// TwinCAT 3 PLC project UnitTests
// Title: Unit Tests for Simple Unit test Lib
// Company: Red Rock Controls Limited
// Author: R Christopher
// ProjectVersion: 1.0.0.0
// ProgramVersion: 3.1.4023.0
// libraries:
//   Tc2_Standard, * (Beckhoff Automation GmbH)
//   Tc2_System, * (Beckhoff Automation GmbH)
//   Tc3_Module, * (Beckhoff Automation GmbH)
//   tcl_SimpleUnitTestLibrary, * (Red Rock Controls Limited)
//   tcl_StringUtils, * (Red Rock Controls Limited)
// project tree:
//   / GlobalTextList.TcGTLO, Visualization Manager.TcVMO (not stored), VISU_TASK.TcTTO
//   GVLs/ UnitTests.TcGVL
//   POUs/ PB_TestRunner.TcPOU
//   POUs/Unit Tests/Assertion Tests/ Test_AssertEquals_BLOB_SizeDiffers.TcPOU, Test_AssertEquals_BLOB_TypeClassDiffers.TcPOU, Test_AssertEquals_BLOB_TypeContentDiffers.TcPOU, Test_AssertEquals_BOOL.TcPOU, Test_AssertEquals_BYTE.TcPOU, Test_AssertEquals_DINT.TcPOU, Test_AssertEquals_DWORD.TcPOU, Test_AssertEquals_INT.TcPOU, Test_AssertEquals_INTERFACE.TcPOU, Test_AssertEquals_LINT.TcPOU, Test_AssertEquals_LREAL.TcPOU, Test_AssertEquals_PVOID.TcPOU, Test_AssertEquals_REAL.TcPOU, Test_AssertEquals_STRING.TcPOU, Test_AssertEquals_UDINT.TcPOU, Test_AssertEquals_UINT.TcPOU, Test_AssertEquals_ULINT.TcPOU, Test_AssertEquals_WORD.TcPOU
//   POUs/Unit Tests/Fixtures/ I_ExampleInterface.TcIO, T_ExampleInterfaceImplementation.TcPOU
//   POUs/Unit Tests/Mocks/ T_AssertionListenerMock.TcPOU
//   POUs/Unit Tests/UnitTestBase Tests/ Test_setTestName_setsTestName.TcPOU, T_UnitTestUnderTest.TcPOU
//   Tasks/ MAIN.TcPOU, PlcTask.TcTTO
//   VISUs/ Visualization.TcVIS
// (motion and I/O tree: see PLC project tcl_simpleunittestlibrary)
// real-time tasks:
//   TASK PlcTask: cycle T#10ms, priority 20, ADS port 351
//   TASK VISU_TASK: cycle T#200000us, priority 30, ADS port 350

CONFIGURATION UnitTests
    RESOURCE PLC ON TwinCAT3
        TASK PlcTask(INTERVAL := T#10ms, PRIORITY := 20);
        TASK VISU_TASK(INTERVAL := T#200000us, PRIORITY := 30);
        PROGRAM MAIN WITH PlcTask : MAIN;
        PROGRAM VisuElems_Visu_Prg WITH VISU_TASK : VisuElems.Visu_Prg;
    END_RESOURCE
END_CONFIGURATION

// ---- GVLs/UnitTests.TcGVL
{attribute 'qualified_only'}
VAR_GLOBAL
    TestFrameworkTests : T_TestSuite;

    Test_AssertEquals_BOOL      : Test_AssertEquals_BOOL        (TestSuite := TestFrameworkTests);
    Test_AssertEquals_BYTE      : Test_AssertEquals_BYTE        (TestSuite := TestFrameworkTests);
    Test_AssertEquals_DINT      : Test_AssertEquals_DINT        (TestSuite := TestFrameworkTests);
    Test_AssertEquals_INT       : Test_AssertEquals_INT         (TestSuite := TestFrameworkTests);
    Test_AssertEquals_INTERFACE : Test_AssertEquals_INTERFACE   (TestSuite := TestFrameworkTests);
    Test_AssertEquals_LINT      : Test_AssertEquals_LINT        (TestSuite := TestFrameworkTests);
    Test_AssertEquals_LREAL     : Test_AssertEquals_LREAL       (TestSuite := TestFrameworkTests);
    Test_AssertEquals_PVOID     : Test_AssertEquals_PVOID       (TestSuite := TestFrameworkTests);
    Test_AssertEquals_REAL      : Test_AssertEquals_REAL        (TestSuite := TestFrameworkTests);
    Test_AssertEquals_STRING    : Test_AssertEquals_STRING      (TestSuite := TestFrameworkTests);
    Test_AssertEquals_UDINT     : Test_AssertEquals_UDINT       (TestSuite := TestFrameworkTests);
    Test_AssertEquals_UINT      : Test_AssertEquals_UINT        (TestSuite := TestFrameworkTests);
    Test_AssertEquals_ULINT     : Test_AssertEquals_ULINT       (TestSuite := TestFrameworkTests);  
    Test_AssertEquals_WORD      : Test_AssertEquals_WORD        (TestSuite := TestFrameworkTests);
    Test_AssertEquals_DWORD     : Test_AssertEquals_DWORD       (TestSuite := TestFrameworkTests);
    
    Test_AssertEquals_BLOB_SizeDiffers          : Test_AssertEquals_BLOB_SizeDiffers        (TestSuite := TestFrameworkTests);  
    Test_AssertEquals_BLOB_TypeClassDiffers     : Test_AssertEquals_BLOB_TypeClassDiffers   (TestSuite := TestFrameworkTests);
    Test_AssertEquals_BLOB_TypeContentDiffers   : Test_AssertEquals_BLOB_TypeContentDiffers (TestSuite := TestFrameworkTests);
    
    Test_setTestName_setsTestName : Test_setTestName_setsTestName (TestSuite := TestFrameworkTests);


END_VAR

// ---- POUs/Unit Tests/Fixtures/I_ExampleInterface.TcIO
INTERFACE I_ExampleInterface EXTENDS __SYSTEM.IQueryInterface

END_INTERFACE

// ---- Tasks/MAIN.TcPOU
PROGRAM MAIN
VAR
END_VAR

PB_TestRunner();

END_PROGRAM

// ---- POUs/PB_TestRunner.TcPOU
PROGRAM PB_TestRunner
VAR
    Init : BOOL := TRUE;
    TestRunner : T_TestRunner;
END_VAR

IF Init THEN
    TestRunner.AddTestSuite(UnitTests.TestFrameworkTests);
    Init := FALSE;
END_IF

TestRunner();

END_PROGRAM

// ---- POUs/Unit Tests/Assertion Tests/Test_AssertEquals_BOOL.TcPOU
FUNCTION_BLOCK Test_AssertEquals_BOOL EXTENDS T_UnitTestBase
VAR
    AssertionUnderTest : T_Assertion(AssertionListenerMock);
    AssertionListenerMock : T_AssertionListenerMock;
    BOOL_Variable : BOOL := FALSE;
END_VAR

// Initialise the classes under test (may be repaeting the tests)...
AssertionListenerMock.fb_Init(
    bInitRetains      := FALSE,
	bInCopyCode       := FALSE);
AssertionUnderTest.fb_Init(
    bInitRetains      := FALSE,
	bInCopyCode       := FALSE,
    AssertionListener := AssertionListenerMock);

// Test the assertion...
AssertionUnderTest.AssertEquals_BOOL(
    Expected := TRUE,
    Actual   := BOOL_Variable,
    VariableName := 'BOOL_Variable');
    
// Check the assertion worked...    
Assertion.AssertEquals_BOOL(
    Expected := TRUE,
    Actual   := AssertionListenerMock.AssertionFailed,
    VariableName := 'AssertionListenerMock.AssertionFailed');

// Check the assertion messages...    
Assertion.AssertEquals_STRING(
    Expected := 'AssertEquals_BOOL failed in AssertionListenerMock: Value "BOOL_Variable"',
    Actual   := AssertionListenerMock.AssertionMessage,
    VariableName := 'AssertionListenerMock.AssertionMessage');

Assertion.AssertEquals_STRING(
    Expected := '  Expected = TRUE',
    Actual   := AssertionListenerMock.ExpectedAsString,
    VariableName := 'AssertionListenerMock.ExpectedAsString');

Assertion.AssertEquals_STRING(
    Expected := '  Actual   = FALSE',
    Actual   := AssertionListenerMock.ActualAsString,
    VariableName := 'AssertionListenerMock.ActualAsString');

TestFinished();

END_FUNCTION_BLOCK

// ---- POUs/Unit Tests/Mocks/T_AssertionListenerMock.TcPOU
{attribute 'reflection'}
FUNCTION_BLOCK T_AssertionListenerMock IMPLEMENTS I_AssertionListener
VAR
    {attribute 'instance-path'} 
    {attribute 'no_init'}
    _FullTestName : T_MaxString; // Automatically initialised with the full name of the instance
    _TestName : T_MaxString; 
    _AssertionFailed  : BOOL;
    _AssertionMessage : T_MaxString;
    _ExpectedAsString : T_MaxString;
    _ActualAsString   : T_MaxString;
END_VAR

PROPERTY ActualAsString : T_MaxString
GET
ActualAsString := _ActualAsString;
END_GET
SET
_ActualAsString := ActualAsString;
END_SET
END_PROPERTY

PROPERTY AssertionFailed : BOOL
GET
AssertionFailed := _AssertionFailed;
END_GET
SET
_AssertionFailed := AssertionFailed;
END_SET
END_PROPERTY

PROPERTY AssertionMessage : T_MaxString
GET
AssertionMessage := _AssertionMessage;
END_GET
SET
_AssertionMessage := AssertionMessage;
END_SET
END_PROPERTY

PROPERTY ExpectedAsString : T_MaxString
GET
ExpectedAsString := _ExpectedAsString;
END_GET
SET
_ExpectedAsString := ExpectedAsString;
END_SET
END_PROPERTY

METHOD OnAssertionFailed
VAR_INPUT
    AssertionMessage : T_MaxString;
    ExpectedAsString : T_MaxString;
    ActualAsString   : T_MaxString;
END_VAR
_AssertionFailed   := TRUE;
_AssertionMessage  := AssertionMessage;
_ExpectedAsString := ExpectedAsString;
_ActualAsString := ActualAsString;
END_METHOD

PROPERTY TestName : Tc2_System.T_MaxString
GET
VAR_INST
    StringSplitter : T_StringSplitter;
END_VAR
IF _TestName = '' THEN
   
    StringSplitter.Init(
        Str := _FullTestName,
        Delim1 := '.',
        Delim2 := '');
    
    WHILE StringSplitter.HasMore() DO
        _TestName := StringSplitter.GetNext(); // to get last sub-section
    END_WHILE
   
END_IF

TestName := _TestName;
END_GET
END_PROPERTY

END_FUNCTION_BLOCK

// ---- POUs/Unit Tests/Assertion Tests/Test_AssertEquals_BYTE.TcPOU
FUNCTION_BLOCK Test_AssertEquals_BYTE EXTENDS T_UnitTestBase
VAR
    AssertionUnderTest : T_Assertion(AssertionListenerMock);
    AssertionListenerMock : T_AssertionListenerMock;
    BYTE_Variable : BYTE := 123;
END_VAR

// Initialise the classes under test (may be repaeting the tests)...
AssertionListenerMock.fb_Init(
    bInitRetains      := FALSE,
	bInCopyCode       := FALSE);
AssertionUnderTest.fb_Init(
    bInitRetains      := FALSE,
	bInCopyCode       := FALSE,
    AssertionListener := AssertionListenerMock);

// Test the assertion...
AssertionUnderTest.AssertEquals_BYTE(
    Expected := 234,
    Actual   := BYTE_Variable,
    VariableName := 'BYTE_Variable');
 
// Check the assertion worked...    
Assertion.AssertEquals_BOOL(
    Expected := TRUE,
    Actual   := AssertionListenerMock.AssertionFailed,
    VariableName := 'AssertionListenerMock.AssertionFailed');

// Check the assertion messages...    
Assertion.AssertEquals_STRING(
    Expected := 'AssertEquals_BYTE failed in AssertionListenerMock: Value "BYTE_Variable"',
    Actual   := AssertionListenerMock.AssertionMessage,
    VariableName := 'AssertionListenerMock.AssertionMessage');

Assertion.AssertEquals_STRING(
    Expected := '  Expected = 234',
    Actual   := AssertionListenerMock.ExpectedAsString,
    VariableName := 'AssertionListenerMock.ExpectedAsString');

Assertion.AssertEquals_STRING(
    Expected := '  Actual   = 123',
    Actual   := AssertionListenerMock.ActualAsString,
    VariableName := 'AssertionListenerMock.ActualAsString');

TestFinished();

END_FUNCTION_BLOCK

// ---- POUs/Unit Tests/Assertion Tests/Test_AssertEquals_DINT.TcPOU
FUNCTION_BLOCK Test_AssertEquals_DINT EXTENDS T_UnitTestBase
VAR
    AssertionUnderTest : T_Assertion(AssertionListenerMock);
    AssertionListenerMock : T_AssertionListenerMock;
    DINT_Variable : DINT := 1111;
END_VAR

// Initialise the classes under test (may be repaeting the tests)...
AssertionListenerMock.fb_Init(
    bInitRetains      := FALSE,
	bInCopyCode       := FALSE);
AssertionUnderTest.fb_Init(
    bInitRetains      := FALSE,
	bInCopyCode       := FALSE,
    AssertionListener := AssertionListenerMock);

// Test the assertion...
AssertionUnderTest.AssertEquals_DINT(
    Expected := 2222,
    Actual   := DINT_Variable,
    VariableName := 'DINT_Variable');
    
// Check the assertion worked...    
Assertion.AssertEquals_BOOL(
    Expected := TRUE,
    Actual   := AssertionListenerMock.AssertionFailed,
    VariableName := 'AssertionListenerMock.AssertionFailed');

// Check the assertion messages...    
Assertion.AssertEquals_STRING(
    Expected := 'AssertEquals_DINT failed in AssertionListenerMock: Value "DINT_Variable"',
    Actual   := AssertionListenerMock.AssertionMessage,
    VariableName := 'AssertionListenerMock.AssertionMessage');

Assertion.AssertEquals_STRING(
    Expected := '  Expected = 2222',
    Actual   := AssertionListenerMock.ExpectedAsString,
    VariableName := 'AssertionListenerMock.ExpectedAsString');

Assertion.AssertEquals_STRING(
    Expected := '  Actual   = 1111',
    Actual   := AssertionListenerMock.ActualAsString,
    VariableName := 'AssertionListenerMock.ActualAsString');

TestFinished();

END_FUNCTION_BLOCK

// ---- POUs/Unit Tests/Assertion Tests/Test_AssertEquals_INT.TcPOU
FUNCTION_BLOCK Test_AssertEquals_INT EXTENDS T_UnitTestBase
VAR
    AssertionUnderTest : T_Assertion(AssertionListenerMock);
    AssertionListenerMock : T_AssertionListenerMock;
    INT_Variable : INT := 1111;
END_VAR

// Initialise the classes under test (may be repaeting the tests)...
AssertionListenerMock.fb_Init(
    bInitRetains      := FALSE,
	bInCopyCode       := FALSE);
AssertionUnderTest.fb_Init(
    bInitRetains      := FALSE,
	bInCopyCode       := FALSE,
    AssertionListener := AssertionListenerMock);

// Test the assertion...
AssertionUnderTest.AssertEquals_INT(
    Expected := 2222,
    Actual   := INT_Variable,
    VariableName := 'INT_Variable');
 
// Check the assertion worked...    
Assertion.AssertEquals_BOOL(
    Expected := TRUE,
    Actual   := AssertionListenerMock.AssertionFailed,
    VariableName := 'AssertionListenerMock.AssertionFailed');

// Check the assertion messages...    
Assertion.AssertEquals_STRING(
    Expected := 'AssertEquals_INT failed in AssertionListenerMock: Value "INT_Variable"',
    Actual   := AssertionListenerMock.AssertionMessage,
    VariableName := 'AssertionListenerMock.AssertionMessage');

Assertion.AssertEquals_STRING(
    Expected := '  Expected = 2222',
    Actual   := AssertionListenerMock.ExpectedAsString,
    VariableName := 'AssertionListenerMock.ExpectedAsString');

Assertion.AssertEquals_STRING(
    Expected := '  Actual   = 1111',
    Actual   := AssertionListenerMock.ActualAsString,
    VariableName := 'AssertionListenerMock.ActualAsString');

TestFinished();

END_FUNCTION_BLOCK

// ---- POUs/Unit Tests/Assertion Tests/Test_AssertEquals_INTERFACE.TcPOU
FUNCTION_BLOCK Test_AssertEquals_INTERFACE EXTENDS T_UnitTestBase
VAR
    AssertionUnderTest : T_Assertion(AssertionListenerMock);
    AssertionListenerMock : T_AssertionListenerMock;
    
    ExampleInterfaceImplementation1   : T_ExampleInterfaceImplementation;
    INTERFACE_Variable1 : I_ExampleInterface := ExampleInterfaceImplementation1;
    
    ExampleInterfaceImplementation2   : T_ExampleInterfaceImplementation;
    INTERFACE_Variable2 : I_ExampleInterface := ExampleInterfaceImplementation2;
END_VAR

// Initialise the classes under test (may be repaeting the tests)...
AssertionListenerMock.fb_Init(
    bInitRetains      := FALSE,
	bInCopyCode       := FALSE);
AssertionUnderTest.fb_Init(
    bInitRetains      := FALSE,
	bInCopyCode       := FALSE,
    AssertionListener := AssertionListenerMock);

// Test the assertion...
AssertionUnderTest.AssertEquals_INTERFACE(
    Expected := INTERFACE_Variable1,
    Actual   := INTERFACE_Variable2,
    VariableName := 'INTERFACE_Variable2'); 
    
// Check the assertion worked...    
Assertion.AssertEquals_BOOL(
    Expected := TRUE,
    Actual   := AssertionListenerMock.AssertionFailed,
    VariableName := 'AssertionListenerMock.AssertionFailed');

// Check the assertion messages...    
Assertion.AssertEquals_STRING(
    Expected := 'AssertEquals_INTERFACE failed in AssertionListenerMock: Value "INTERFACE_Variable2"',
    Actual   := AssertionListenerMock.AssertionMessage,
    VariableName := 'AssertionListenerMock.AssertionMessage');

Assertion.AssertEquals_STRING(
    Expected := '  Interfaces Differ',
    Actual   := AssertionListenerMock.ExpectedAsString,
    VariableName := 'AssertionListenerMock.ExpectedAsString');

Assertion.AssertEquals_STRING(
    Expected := '',
    Actual   := AssertionListenerMock.ActualAsString,
    VariableName := 'AssertionListenerMock.ActualAsString');

TestFinished();

END_FUNCTION_BLOCK

// ---- POUs/Unit Tests/Fixtures/T_ExampleInterfaceImplementation.TcPOU
FUNCTION_BLOCK T_ExampleInterfaceImplementation IMPLEMENTS I_ExampleInterface
VAR_INPUT
END_VAR
VAR_OUTPUT
END_VAR
VAR
END_VAR

END_FUNCTION_BLOCK

// ---- POUs/Unit Tests/Assertion Tests/Test_AssertEquals_LINT.TcPOU
FUNCTION_BLOCK Test_AssertEquals_LINT EXTENDS T_UnitTestBase
VAR
    AssertionUnderTest : T_Assertion(AssertionListenerMock);
    AssertionListenerMock : T_AssertionListenerMock;
    LINT_Variable : LINT := 1111;
END_VAR

// Initialise the classes under test (may be repaeting the tests)...
AssertionListenerMock.fb_Init(
    bInitRetains      := FALSE,
	bInCopyCode       := FALSE);
AssertionUnderTest.fb_Init(
    bInitRetains      := FALSE,
	bInCopyCode       := FALSE,
    AssertionListener := AssertionListenerMock);

// Test the assertion...
AssertionUnderTest.AssertEquals_LINT(
    Expected := 2222,
    Actual   := LINT_Variable,
    VariableName := 'LINT_Variable');
 
    
// Check the assertion worked...    
Assertion.AssertEquals_BOOL(
    Expected := TRUE,
    Actual   := AssertionListenerMock.AssertionFailed,
    VariableName := 'AssertionListenerMock.AssertionFailed');

// Check the assertion messages...    
Assertion.AssertEquals_STRING(
    Expected := 'AssertEquals_LINT failed in AssertionListenerMock: Value "LINT_Variable"',
    Actual   := AssertionListenerMock.AssertionMessage,
    VariableName := 'AssertionListenerMock.AssertionMessage');

Assertion.AssertEquals_STRING(
    Expected := '  Expected = 2222',
    Actual   := AssertionListenerMock.ExpectedAsString,
    VariableName := 'AssertionListenerMock.ExpectedAsString');

Assertion.AssertEquals_STRING(
    Expected := '  Actual   = 1111',
    Actual   := AssertionListenerMock.ActualAsString,
    VariableName := 'AssertionListenerMock.ActualAsString');

TestFinished();

END_FUNCTION_BLOCK

// ---- POUs/Unit Tests/Assertion Tests/Test_AssertEquals_LREAL.TcPOU
FUNCTION_BLOCK Test_AssertEquals_LREAL EXTENDS T_UnitTestBase
VAR
    AssertionUnderTest : T_Assertion(AssertionListenerMock);
    AssertionListenerMock : T_AssertionListenerMock;
    LREAL_Variable : LREAL := 1.111;
END_VAR

// Initialise the classes under test (may be repaeting the tests)...
AssertionListenerMock.fb_Init(
    bInitRetains      := FALSE,
	bInCopyCode       := FALSE);
AssertionUnderTest.fb_Init(
    bInitRetains      := FALSE,
	bInCopyCode       := FALSE,
    AssertionListener := AssertionListenerMock);

// Test the assertion...
AssertionUnderTest.AssertEquals_LREAL(
    Expected := 2.222,
    Actual   := LREAL_Variable,
    Delta    := 0.001,
    VariableName := 'LREAL_Variable');
   
// Check the assertion worked...    
Assertion.AssertEquals_BOOL(
    Expected := TRUE,
    Actual   := AssertionListenerMock.AssertionFailed,
    VariableName := 'AssertionListenerMock.AssertionFailed');

// Check the assertion messages...    
Assertion.AssertEquals_STRING(
    Expected := 'AssertEquals_LREAL failed in AssertionListenerMock: Value "LREAL_Variable"',
    Actual   := AssertionListenerMock.AssertionMessage,
    VariableName := 'AssertionListenerMock.AssertionMessage');

Assertion.AssertEquals_STRING(
    Expected := '  Expected = 2.222000',
    Actual   := AssertionListenerMock.ExpectedAsString,
    VariableName := 'AssertionListenerMock.ExpectedAsString');

Assertion.AssertEquals_STRING(
    Expected := '  Actual   = 1.111000',
    Actual   := AssertionListenerMock.ActualAsString,
    VariableName := 'AssertionListenerMock.ActualAsString');

TestFinished();

END_FUNCTION_BLOCK

// ---- POUs/Unit Tests/Assertion Tests/Test_AssertEquals_PVOID.TcPOU
FUNCTION_BLOCK Test_AssertEquals_PVOID EXTENDS T_UnitTestBase
VAR
    AssertionUnderTest : T_Assertion(AssertionListenerMock);
    AssertionListenerMock : T_AssertionListenerMock;
    PVOID_Variable : PVOID := 1111;
END_VAR

// Initialise the classes under test (may be repaeting the tests)...
AssertionListenerMock.fb_Init(
    bInitRetains      := FALSE,
	bInCopyCode       := FALSE);
AssertionUnderTest.fb_Init(
    bInitRetains      := FALSE,
	bInCopyCode       := FALSE,
    AssertionListener := AssertionListenerMock);

// Test the assertion...
AssertionUnderTest.AssertEquals_PVOID(
    Expected := 2222,
    Actual   := PVOID_Variable,
    VariableName := 'PVOID_Variable'); 
    
// Check the assertion worked...    
Assertion.AssertEquals_BOOL(
    Expected := TRUE,
    Actual   := AssertionListenerMock.AssertionFailed,
    VariableName := 'AssertionListenerMock.AssertionFailed');

// Check the assertion messages...    
Assertion.AssertEquals_STRING(
    Expected := 'AssertEquals_PVOID failed in AssertionListenerMock: Value "PVOID_Variable"',
    Actual   := AssertionListenerMock.AssertionMessage,
    VariableName := 'AssertionListenerMock.AssertionMessage');

Assertion.AssertEquals_STRING(
    Expected := '  Expected = 2222',
    Actual   := AssertionListenerMock.ExpectedAsString,
    VariableName := 'AssertionListenerMock.ExpectedAsString');

Assertion.AssertEquals_STRING(
    Expected := '  Actual   = 1111',
    Actual   := AssertionListenerMock.ActualAsString,
    VariableName := 'AssertionListenerMock.ActualAsString');

TestFinished();

END_FUNCTION_BLOCK

// ---- POUs/Unit Tests/Assertion Tests/Test_AssertEquals_REAL.TcPOU
FUNCTION_BLOCK Test_AssertEquals_REAL EXTENDS T_UnitTestBase
VAR
    AssertionUnderTest : T_Assertion(AssertionListenerMock);
    AssertionListenerMock : T_AssertionListenerMock;
    REAL_Variable : REAL := 1.111;
END_VAR

// Initialise the classes under test (may be repaeting the tests)...
AssertionListenerMock.fb_Init(
    bInitRetains      := FALSE,
	bInCopyCode       := FALSE);
AssertionUnderTest.fb_Init(
    bInitRetains      := FALSE,
	bInCopyCode       := FALSE,
    AssertionListener := AssertionListenerMock);

// Test the assertion...
AssertionUnderTest.AssertEquals_REAL(
    Expected := 2.222,
    Actual   := REAL_Variable,
    Delta    := 0.001,
    VariableName := 'REAL_Variable');
  
// Check the assertion worked...    
Assertion.AssertEquals_BOOL(
    Expected := TRUE,
    Actual   := AssertionListenerMock.AssertionFailed,
    VariableName := 'AssertionListenerMock.AssertionFailed');

// Check the assertion messages...    
Assertion.AssertEquals_STRING(
    Expected := 'AssertEquals_REAL failed in AssertionListenerMock: Value "REAL_Variable"',
    Actual   := AssertionListenerMock.AssertionMessage,
    VariableName := 'AssertionListenerMock.AssertionMessage');

Assertion.AssertEquals_STRING(
    Expected := '  Expected = 2.222000',
    Actual   := AssertionListenerMock.ExpectedAsString,
    VariableName := 'AssertionListenerMock.ExpectedAsString');

Assertion.AssertEquals_STRING(
    Expected := '  Actual   = 1.111000',
    Actual   := AssertionListenerMock.ActualAsString,
    VariableName := 'AssertionListenerMock.ActualAsString');

TestFinished();

END_FUNCTION_BLOCK

// ---- POUs/Unit Tests/Assertion Tests/Test_AssertEquals_STRING.TcPOU
FUNCTION_BLOCK Test_AssertEquals_STRING EXTENDS T_UnitTestBase
VAR
    AssertionUnderTest : T_Assertion(AssertionListenerMock);
    AssertionListenerMock : T_AssertionListenerMock;
    STRING_Variable : STRING := 'Cucumber';
END_VAR

// Initialise the classes under test (may be repaeting the tests)...
AssertionListenerMock.fb_Init(
    bInitRetains      := FALSE,
	bInCopyCode       := FALSE);
AssertionUnderTest.fb_Init(
    bInitRetains      := FALSE,
	bInCopyCode       := FALSE,
    AssertionListener := AssertionListenerMock);

// Test the assertion...
AssertionUnderTest.AssertEquals_STRING(
    Expected := 'Radish',
    Actual   := STRING_Variable,
    VariableName := 'STRING_Variable'); 
    
// Check the assertion worked...    
Assertion.AssertEquals_BOOL(
    Expected := TRUE,
    Actual   := AssertionListenerMock.AssertionFailed,
    VariableName := 'AssertionListenerMock.AssertionFailed');

// Check the assertion messages...    
Assertion.AssertEquals_STRING(
    Expected := 'AssertEquals_STRING failed in AssertionListenerMock: Value "STRING_Variable"',
    Actual   := AssertionListenerMock.AssertionMessage,
    VariableName := 'AssertionListenerMock.AssertionMessage');

Assertion.AssertEquals_STRING(
    Expected := '  Expected = Radish',
    Actual   := AssertionListenerMock.ExpectedAsString,
    VariableName := 'AssertionListenerMock.ExpectedAsString');

Assertion.AssertEquals_STRING(
    Expected := '  Actual   = Cucumber',
    Actual   := AssertionListenerMock.ActualAsString,
    VariableName := 'AssertionListenerMock.ActualAsString');

TestFinished();

END_FUNCTION_BLOCK

// ---- POUs/Unit Tests/Assertion Tests/Test_AssertEquals_UDINT.TcPOU
FUNCTION_BLOCK Test_AssertEquals_UDINT EXTENDS T_UnitTestBase
VAR
    AssertionUnderTest : T_Assertion(AssertionListenerMock);
    AssertionListenerMock : T_AssertionListenerMock;
    UDINT_Variable : UDINT := 1111;
END_VAR

// Initialise the classes under test (may be repaeting the tests)...
AssertionListenerMock.fb_Init(
    bInitRetains      := FALSE,
	bInCopyCode       := FALSE);
AssertionUnderTest.fb_Init(
    bInitRetains      := FALSE,
	bInCopyCode       := FALSE,
    AssertionListener := AssertionListenerMock);

// Test the assertion...
AssertionUnderTest.AssertEquals_UDINT(
    Expected := 2222,
    Actual   := UDINT_Variable,
    VariableName := 'UDINT_Variable');
    
// Check the assertion worked...    
Assertion.AssertEquals_BOOL(
    Expected := TRUE,
    Actual   := AssertionListenerMock.AssertionFailed,
    VariableName := 'AssertionListenerMock.AssertionFailed');

// Check the assertion messages...    
Assertion.AssertEquals_STRING(
    Expected := 'AssertEquals_UDINT failed in AssertionListenerMock: Value "UDINT_Variable"',
    Actual   := AssertionListenerMock.AssertionMessage,
    VariableName := 'AssertionListenerMock.AssertionMessage');

Assertion.AssertEquals_STRING(
    Expected := '  Expected = 2222',
    Actual   := AssertionListenerMock.ExpectedAsString,
    VariableName := 'AssertionListenerMock.ExpectedAsString');

Assertion.AssertEquals_STRING(
    Expected := '  Actual   = 1111',
    Actual   := AssertionListenerMock.ActualAsString,
    VariableName := 'AssertionListenerMock.ActualAsString');

TestFinished();

END_FUNCTION_BLOCK

// ---- POUs/Unit Tests/Assertion Tests/Test_AssertEquals_UINT.TcPOU
FUNCTION_BLOCK Test_AssertEquals_UINT EXTENDS T_UnitTestBase
VAR
    AssertionUnderTest : T_Assertion(AssertionListenerMock);
    AssertionListenerMock : T_AssertionListenerMock;
    UINT_Variable : UINT := 1111;
END_VAR

// Initialise the classes under test (may be repaeting the tests)...
AssertionListenerMock.fb_Init(
    bInitRetains      := FALSE,
	bInCopyCode       := FALSE);
AssertionUnderTest.fb_Init(
    bInitRetains      := FALSE,
	bInCopyCode       := FALSE,
    AssertionListener := AssertionListenerMock);

// Test the assertion...
AssertionUnderTest.AssertEquals_UINT(
    Expected := 2222,
    Actual   := UINT_Variable,
    VariableName := 'UINT_Variable');
   
// Check the assertion worked...    
Assertion.AssertEquals_BOOL(
    Expected := TRUE,
    Actual   := AssertionListenerMock.AssertionFailed,
    VariableName := 'AssertionListenerMock.AssertionFailed');

// Check the assertion messages...    
Assertion.AssertEquals_STRING(
    Expected := 'AssertEquals_UINT failed in AssertionListenerMock: Value "UINT_Variable"',
    Actual   := AssertionListenerMock.AssertionMessage,

    VariableName := 'AssertionListenerMock.AssertionMessage');

Assertion.AssertEquals_STRING(
    Expected := '  Expected = 2222',
    Actual   := AssertionListenerMock.ExpectedAsString,
    VariableName := 'AssertionListenerMock.ExpectedAsString');

Assertion.AssertEquals_STRING(
    Expected := '  Actual   = 1111',
    Actual   := AssertionListenerMock.ActualAsString,
    VariableName := 'AssertionListenerMock.ActualAsString');

TestFinished();

END_FUNCTION_BLOCK

// ---- POUs/Unit Tests/Assertion Tests/Test_AssertEquals_ULINT.TcPOU
FUNCTION_BLOCK Test_AssertEquals_ULINT EXTENDS T_UnitTestBase
VAR
    AssertionUnderTest : T_Assertion(AssertionListenerMock);
    AssertionListenerMock : T_AssertionListenerMock;
    ULINT_Variable : ULINT := 1111;
END_VAR

// Initialise the classes under test (may be repaeting the tests)...
AssertionListenerMock.fb_Init(
    bInitRetains      := FALSE,
	bInCopyCode       := FALSE);
AssertionUnderTest.fb_Init(
    bInitRetains      := FALSE,
	bInCopyCode       := FALSE,
    AssertionListener := AssertionListenerMock);

// Test the assertion...
AssertionUnderTest.AssertEquals_ULINT(
    Expected := 2222,
    Actual   := ULINT_Variable,
    VariableName := 'ULINT_Variable');
   
// Check the assertion worked...    
Assertion.AssertEquals_BOOL(
    Expected := TRUE,
    Actual   := AssertionListenerMock.AssertionFailed,
    VariableName := 'AssertionListenerMock.AssertionFailed');

// Check the assertion messages...    
Assertion.AssertEquals_STRING(
    Expected := 'AssertEquals_ULINT failed in AssertionListenerMock: Value "ULINT_Variable"',
    Actual   := AssertionListenerMock.AssertionMessage,
    VariableName := 'AssertionListenerMock.AssertionMessage');

Assertion.AssertEquals_STRING(
    Expected := '  Expected = 2222',
    Actual   := AssertionListenerMock.ExpectedAsString,
    VariableName := 'AssertionListenerMock.ExpectedAsString');

Assertion.AssertEquals_STRING(
    Expected := '  Actual   = 1111',
    Actual   := AssertionListenerMock.ActualAsString,
    VariableName := 'AssertionListenerMock.ActualAsString');

TestFinished();

END_FUNCTION_BLOCK

// ---- POUs/Unit Tests/Assertion Tests/Test_AssertEquals_WORD.TcPOU
FUNCTION_BLOCK Test_AssertEquals_WORD EXTENDS T_UnitTestBase
VAR
    AssertionUnderTest : T_Assertion(AssertionListenerMock);
    AssertionListenerMock : T_AssertionListenerMock;
    WORD_Variable : WORD;
END_VAR

// Initialise the classes under test (may be repaeting the tests)...
AssertionListenerMock.fb_Init(
    bInitRetains      := FALSE,
	bInCopyCode       := FALSE);
AssertionUnderTest.fb_Init(
    bInitRetains      := FALSE,
	bInCopyCode       := FALSE,
    AssertionListener := AssertionListenerMock);

// Test the assertion...
WORD_Variable := 1111;

AssertionUnderTest.AssertEquals_WORD(
    Expected := 2222, // deliberately different to test the assertion
    Actual   := WORD_Variable,
    VariableName := 'WORD_Variable');
 
// Check the assertion worked...    
Assertion.AssertEquals_BOOL(
    Expected := TRUE,
    Actual   := AssertionListenerMock.AssertionFailed,
    VariableName := 'AssertionListenerMock.AssertionFailed');

// Check the assertion messages...    
Assertion.AssertEquals_STRING(
    Expected := 'AssertEquals_WORD failed in AssertionListenerMock: Value "WORD_Variable"',
    Actual   := AssertionListenerMock.AssertionMessage,
    VariableName := 'AssertionListenerMock.AssertionMessage');

Assertion.AssertEquals_STRING(
    Expected := '  Expected = 2222',
    Actual   := AssertionListenerMock.ExpectedAsString,
    VariableName := 'AssertionListenerMock.ExpectedAsString');

Assertion.AssertEquals_STRING(
    Expected := '  Actual   = 1111',
    Actual   := AssertionListenerMock.ActualAsString,
    VariableName := 'AssertionListenerMock.ActualAsString');


TestFinished();

END_FUNCTION_BLOCK

// ---- POUs/Unit Tests/Assertion Tests/Test_AssertEquals_DWORD.TcPOU
FUNCTION_BLOCK Test_AssertEquals_DWORD EXTENDS T_UnitTestBase
VAR
    AssertionUnderTest : T_Assertion(AssertionListenerMock);
    AssertionListenerMock : T_AssertionListenerMock;
    DWORD_Variable : DWORD;
END_VAR

// Initialise the classes under test (may be repaeting the tests)...
AssertionListenerMock.fb_Init(
    bInitRetains      := FALSE,
	bInCopyCode       := FALSE);
AssertionUnderTest.fb_Init(
    bInitRetains      := FALSE,
	bInCopyCode       := FALSE,
    AssertionListener := AssertionListenerMock);

// Test the assertion...
DWORD_Variable := 1111;

AssertionUnderTest.AssertEquals_DWORD(
    Expected := 2222, // deliberately different to test the assertion
    Actual   := DWORD_Variable,
    VariableName := 'DWORD_Variable');
 
    
// Check the assertion worked...    
Assertion.AssertEquals_BOOL(
    Expected := TRUE,
    Actual   := AssertionListenerMock.AssertionFailed,
    VariableName := 'AssertionListenerMock.AssertionFailed');

// Check the assertion messages...    
Assertion.AssertEquals_STRING(
    Expected := 'AssertEquals_DWORD failed in AssertionListenerMock: Value "DWORD_Variable"',
    Actual   := AssertionListenerMock.AssertionMessage,
    VariableName := 'AssertionListenerMock.AssertionMessage');

Assertion.AssertEquals_STRING(
    Expected := '  Expected = 2222',
    Actual   := AssertionListenerMock.ExpectedAsString,
    VariableName := 'AssertionListenerMock.ExpectedAsString');

Assertion.AssertEquals_STRING(
    Expected := '  Actual   = 1111',
    Actual   := AssertionListenerMock.ActualAsString,
    VariableName := 'AssertionListenerMock.ActualAsString');

TestFinished();

END_FUNCTION_BLOCK

// ---- POUs/Unit Tests/Assertion Tests/Test_AssertEquals_BLOB_SizeDiffers.TcPOU
FUNCTION_BLOCK Test_AssertEquals_BLOB_SizeDiffers EXTENDS T_UnitTestBase
VAR
    AssertionUnderTest : T_Assertion(AssertionListenerMock);
    AssertionListenerMock : T_AssertionListenerMock;
    BYTE_Variable : BYTE := 123;
    WORD_Variable : WORD := 456;
END_VAR

// Initialise the classes under test (may be repaeting the tests)...
AssertionListenerMock.fb_Init(
    bInitRetains      := FALSE,
	bInCopyCode       := FALSE);
AssertionUnderTest.fb_Init(
    bInitRetains      := FALSE,
	bInCopyCode       := FALSE,
    AssertionListener := AssertionListenerMock);

// Test the assertion...
AssertionUnderTest.AssertEquals_BLOB(
    Expected := BYTE_Variable,
    Actual   := WORD_Variable,
    VariableName := 'WORD_VariableAsBlob');
 
    
// Check the assertion worked...    
Assertion.AssertEquals_BOOL(
    Expected := TRUE,
    Actual   := AssertionListenerMock.AssertionFailed,
    VariableName := 'AssertionListenerMock.AssertionFailed');

// Check the assertion messages...    
Assertion.AssertEquals_STRING(
    Expected := 'AssertEquals_BLOB failed in AssertionListenerMock: Value "Blob.Size"',
    Actual   := AssertionListenerMock.AssertionMessage,
    VariableName := 'AssertionListenerMock.AssertionMessage');

Assertion.AssertEquals_STRING(
    Expected := '  Expected = 1',
    Actual   := AssertionListenerMock.ExpectedAsString,
    VariableName := 'AssertionListenerMock.ExpectedAsString');

Assertion.AssertEquals_STRING(
    Expected := '  Actual   = 2',
    Actual   := AssertionListenerMock.ActualAsString,
    VariableName := 'AssertionListenerMock.ActualAsString');

TestFinished();

END_FUNCTION_BLOCK

// ---- POUs/Unit Tests/Assertion Tests/Test_AssertEquals_BLOB_TypeClassDiffers.TcPOU
FUNCTION_BLOCK Test_AssertEquals_BLOB_TypeClassDiffers EXTENDS T_UnitTestBase
VAR
    AssertionUnderTest : T_Assertion(AssertionListenerMock);
    AssertionListenerMock : T_AssertionListenerMock;
    
    // Sizes are the same, but TypeClass differs...
    INT_Variable  : INT  := 123;
    WORD_Variable : WORD := 123;
END_VAR

// Initialise the classes under test (may be repaeting the tests)...
AssertionListenerMock.fb_Init(
    bInitRetains      := FALSE,
	bInCopyCode       := FALSE);
AssertionUnderTest.fb_Init(
    bInitRetains      := FALSE,
	bInCopyCode       := FALSE,
    AssertionListener := AssertionListenerMock);

// Test the assertion...
AssertionUnderTest.AssertEquals_BLOB(
    Expected := INT_Variable,
    Actual   := WORD_Variable,
    VariableName := 'WORD_VariableAsBlob');
 
// Check the assertion worked...    
Assertion.AssertEquals_BOOL(
    Expected := TRUE,
    Actual   := AssertionListenerMock.AssertionFailed,
    VariableName := 'AssertionListenerMock.AssertionFailed');

// Check the assertion messages...    
Assertion.AssertEquals_STRING(
    Expected := 'AssertEquals_BLOB failed in AssertionListenerMock: Value "Blob.TypeClass"',
    Actual   := AssertionListenerMock.AssertionMessage,
    VariableName := 'AssertionListenerMock.AssertionMessage');

Assertion.AssertEquals_STRING(
    Expected := '  Expected = INT',
    Actual   := AssertionListenerMock.ExpectedAsString,
    VariableName := 'AssertionListenerMock.ExpectedAsString');

Assertion.AssertEquals_STRING(
    Expected := '  Actual   = WORD',
    Actual   := AssertionListenerMock.ActualAsString,
    VariableName := 'AssertionListenerMock.ActualAsString');

TestFinished();

END_FUNCTION_BLOCK

// ---- POUs/Unit Tests/Assertion Tests/Test_AssertEquals_BLOB_TypeContentDiffers.TcPOU
FUNCTION_BLOCK Test_AssertEquals_BLOB_TypeContentDiffers EXTENDS T_UnitTestBase
VAR
    AssertionUnderTest : T_Assertion(AssertionListenerMock);
    AssertionListenerMock : T_AssertionListenerMock;
    
    // Sizes are the same, but TypeClass differs...
    INT_Variable  : WORD := 123;
    WORD_Variable : WORD := 124;
END_VAR

// Initialise the classes under test (may be repaeting the tests)...
AssertionListenerMock.fb_Init(
    bInitRetains      := FALSE,
	bInCopyCode       := FALSE);
AssertionUnderTest.fb_Init(
    bInitRetains      := FALSE,
	bInCopyCode       := FALSE,
    AssertionListener := AssertionListenerMock);

// Test the assertion...
AssertionUnderTest.AssertEquals_BLOB(
    Expected := INT_Variable,
    Actual   := WORD_Variable,
    VariableName := 'WORD_VariableAsBlob');
 
// Check the assertion worked...    
Assertion.AssertEquals_BOOL(
    Expected := TRUE,
    Actual   := AssertionListenerMock.AssertionFailed,
    VariableName := 'AssertionListenerMock.AssertionFailed');

// Check the assertion messages...    
Assertion.AssertEquals_STRING(
    Expected := 'AssertEquals_BLOB failed in AssertionListenerMock: Contents differ',
    Actual   := AssertionListenerMock.AssertionMessage,
    VariableName := 'AssertionListenerMock.AssertionMessage');

Assertion.AssertEquals_STRING(
    Expected := '',
    Actual   := AssertionListenerMock.ExpectedAsString,
    VariableName := 'AssertionListenerMock.ExpectedAsString');

Assertion.AssertEquals_STRING(
    Expected := '',
    Actual   := AssertionListenerMock.ActualAsString,
    VariableName := 'AssertionListenerMock.ActualAsString');

TestFinished();

END_FUNCTION_BLOCK

// ---- POUs/Unit Tests/UnitTestBase Tests/Test_setTestName_setsTestName.TcPOU
FUNCTION_BLOCK Test_setTestName_setsTestName EXTENDS T_UnitTestBase
VAR_INPUT
END_VAR
VAR_OUTPUT
END_VAR
VAR
    UnitTest : T_UnitTestUnderTest(TestSuite := 0); // not added to Test Runner
END_VAR

UnitTest.setTestName();

Assertion.AssertEquals_STRING(
    Expected := 'UnitTest',
    Actual   := UnitTest.TestName,
    VariableName := 'UnitTest.TestName');
    
TestFinished();

END_FUNCTION_BLOCK

// ---- POUs/Unit Tests/UnitTestBase Tests/T_UnitTestUnderTest.TcPOU
FUNCTION_BLOCK T_UnitTestUnderTest EXTENDS T_UnitTestBase
VAR_INPUT
END_VAR
VAR_OUTPUT
END_VAR
VAR
END_VAR

END_FUNCTION_BLOCK

// ---- GlobalTextList.TcGTLO
TEXTLIST GlobalTextList
  346 = 'Checkbox'
  643 = 'Run Sequentially'
END_TEXTLIST

// ---- VISUs/Visualization.TcVIS
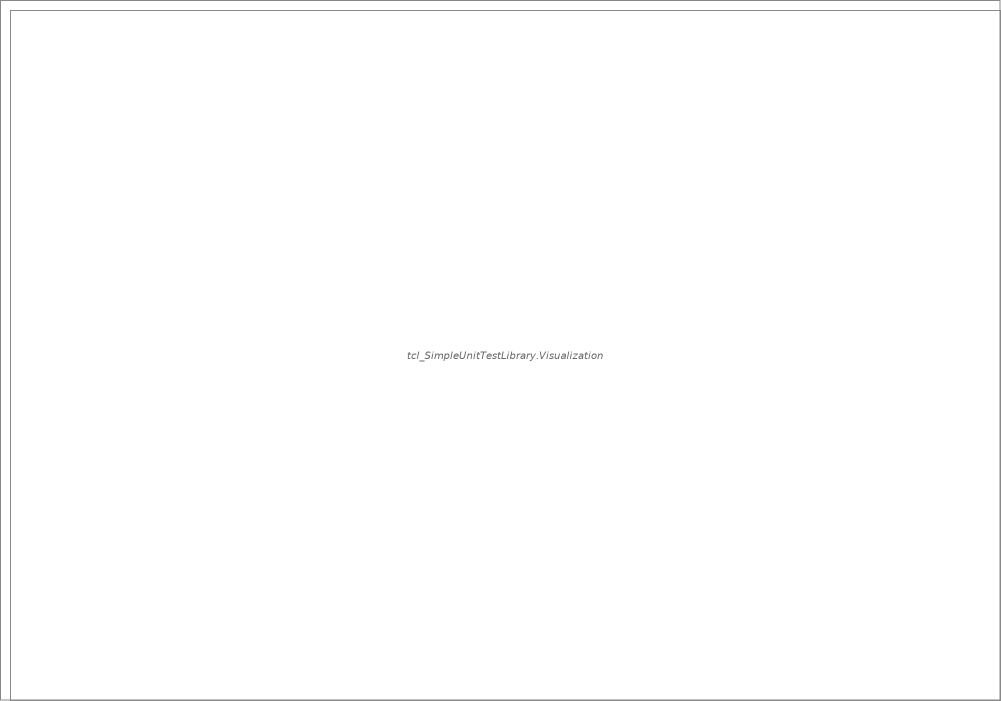
VISUALIZATION Visualization  // 1001x701
    Frame (10,10 991x691)
        shows tcl_SimpleUnitTestLibrary.Visualization(TestRunner := PB_TestRunner.TestRunner)
END_VISUALIZATION
